FUNCTION Convert_DWORD_TO_UDINT : Hresult
VAR_INPUT
	in : DWORD;
	out : REFERENCE TO UDINT;
END_VAR
VAR
	converted : UDINT;
END_VAR

converted := DWORD_TO_UDINT(in);

IF (UDINT_TO_DWORD(converted) <> in) THEN
	Convert_DWORD_TO_UDINT := INCOMPATIBLE;
	RETURN;
END_IF

out := converted;

END_FUNCTION

(* stored: Version 1.1.0.1, ProductVersion 3.1.4024.12
   POU Convert_DWORD_TO_UDINT: Id {96d31378-b2d4-4a60-a4f5-62afa6930bc9}, SpecialFunc None *)
